{attribute 'GeneratedUsingTerminal: KL9900-0057'}
{attribute addProperty BoxType "KL9900-0057"}
{attribute addProperty Id "Channel_1AT %Q*Channel_61FC15360"}
{attribute addProperty CRC "1524632092"}
{attribute addProperty Size "0"}
TYPE KL_5AE00A1C :
STRUCT
	{attribute addProperty Name "Channel_1"}
	Channel_1 : Channel_61FC1536;
END_STRUCT
END_TYPE

(* stored: Version 1.2.0.0, ProductVersion 3.1.4024.9
   DUT KL_5AE00A1C: Id {38f10df5-5f04-41a7-bec0-ac0fdd91dc3b} *)
